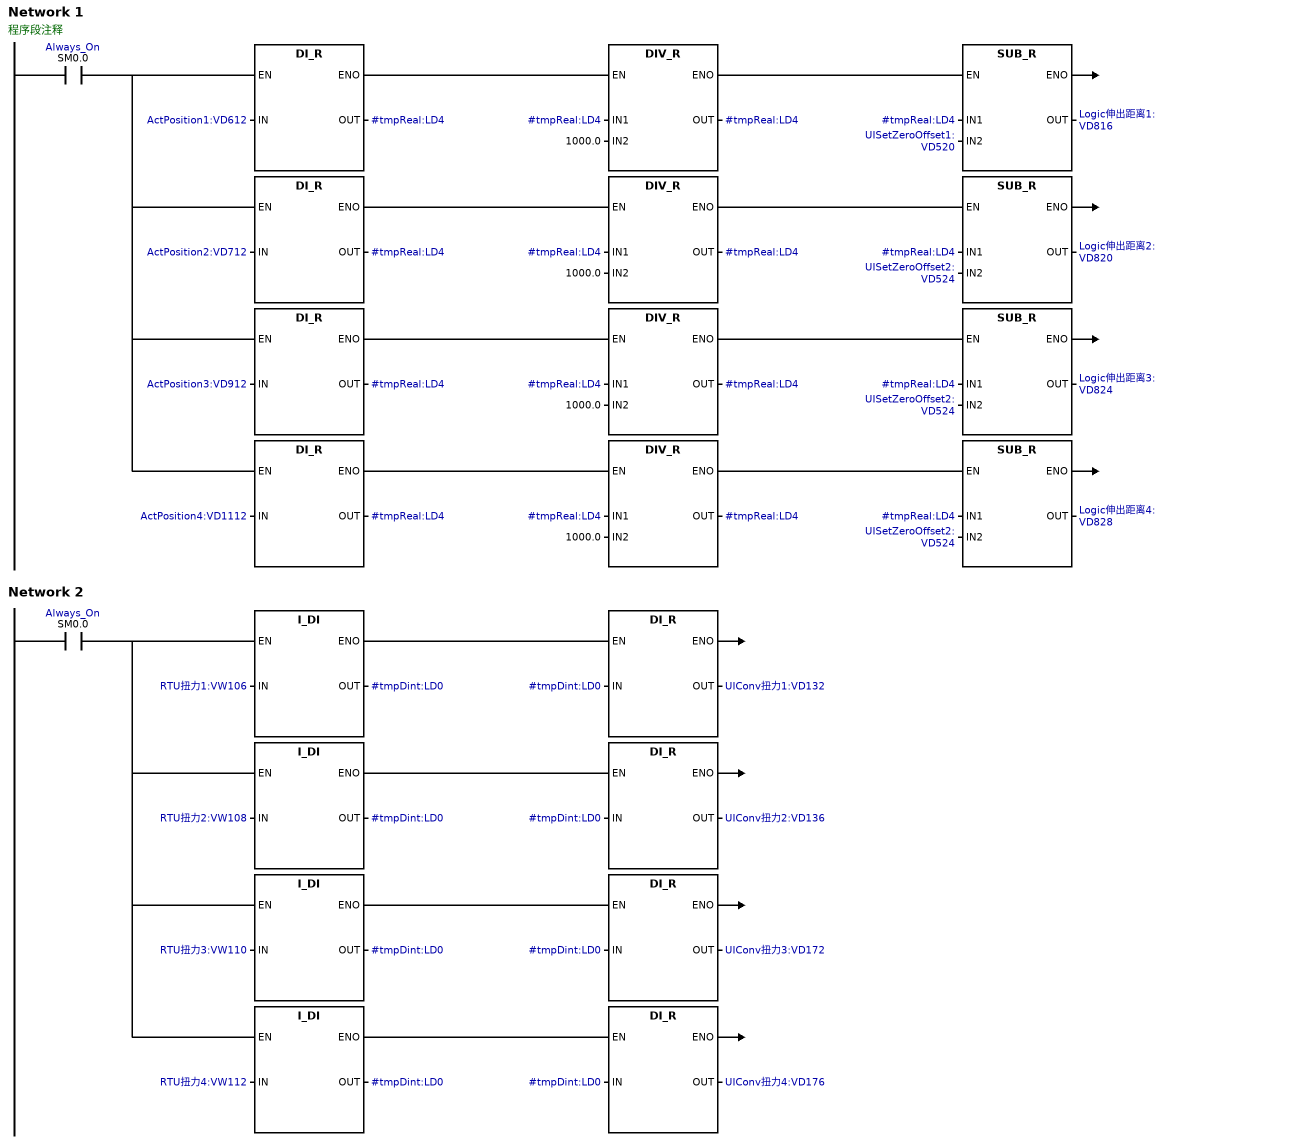
[picture p24: SBR6 networks 1-2]
Network 1
// 程序段注释
LD     Always_On:SM0.0
LPS
DTR    ActPosition1:VD612, #tmpReal:LD4
AENO
/R     1000.0, #tmpReal:LD4
AENO
MOVR   #tmpReal:LD4, Logic伸出距离1:VD816
-R     UISetZeroOffset1:VD520, Logic伸出距离1:VD816
LRD
DTR    ActPosition2:VD712, #tmpReal:LD4
AENO
/R     1000.0, #tmpReal:LD4
AENO
MOVR   #tmpReal:LD4, Logic伸出距离2:VD820
-R     UISetZeroOffset2:VD524, Logic伸出距离2:VD820
LRD
DTR    ActPosition3:VD912, #tmpReal:LD4
AENO
/R     1000.0, #tmpReal:LD4
AENO
MOVR   #tmpReal:LD4, Logic伸出距离3:VD824
-R     UISetZeroOffset2:VD524, Logic伸出距离3:VD824
LPP
DTR    ActPosition4:VD1112, #tmpReal:LD4
AENO
/R     1000.0, #tmpReal:LD4
AENO
MOVR   #tmpReal:LD4, Logic伸出距离4:VD828
-R     UISetZeroOffset2:VD524, Logic伸出距离4:VD828
Network 2
LD     Always_On:SM0.0
LPS
ITD    RTU扭力1:VW106, #tmpDint:LD0
AENO
DTR    #tmpDint:LD0, UIConv扭力1:VD132
LRD
ITD    RTU扭力2:VW108, #tmpDint:LD0
AENO
DTR    #tmpDint:LD0, UIConv扭力2:VD136
LRD
ITD    RTU扭力3:VW110, #tmpDint:LD0
AENO
DTR    #tmpDint:LD0, UIConv扭力3:VD172
LPP
ITD    RTU扭力4:VW112, #tmpDint:LD0
AENO
DTR    #tmpDint:LD0, UIConv扭力4:VD176
END_SUBROUTINE_BLOCK

// SBR7: protected block, not included

// SBR8: protected block, not included

SUBROUTINE_BLOCK XinJiePN:SBR9
TITLE=子程序注释
VAR
tmpSpeed:DWORD;	// LD0 
tmpPos1:DINT;	// LD4 
tmpWarning:WORD;	// LW8 
tmpErr:WORD;	// LW10 
tmpDone:BOOL;	// L12.0 
tmpNotJOD:BOOL;	// L12.1 
tmpPos2:DINT;	// LD13 
tmpReal:REAL;	// LD17 
tmpDint:DINT;	// LD21 
tmpPos3:DINT;	// LD25 
tmpPos4:DINT;	// LD29 
END_VAR
BEGIN
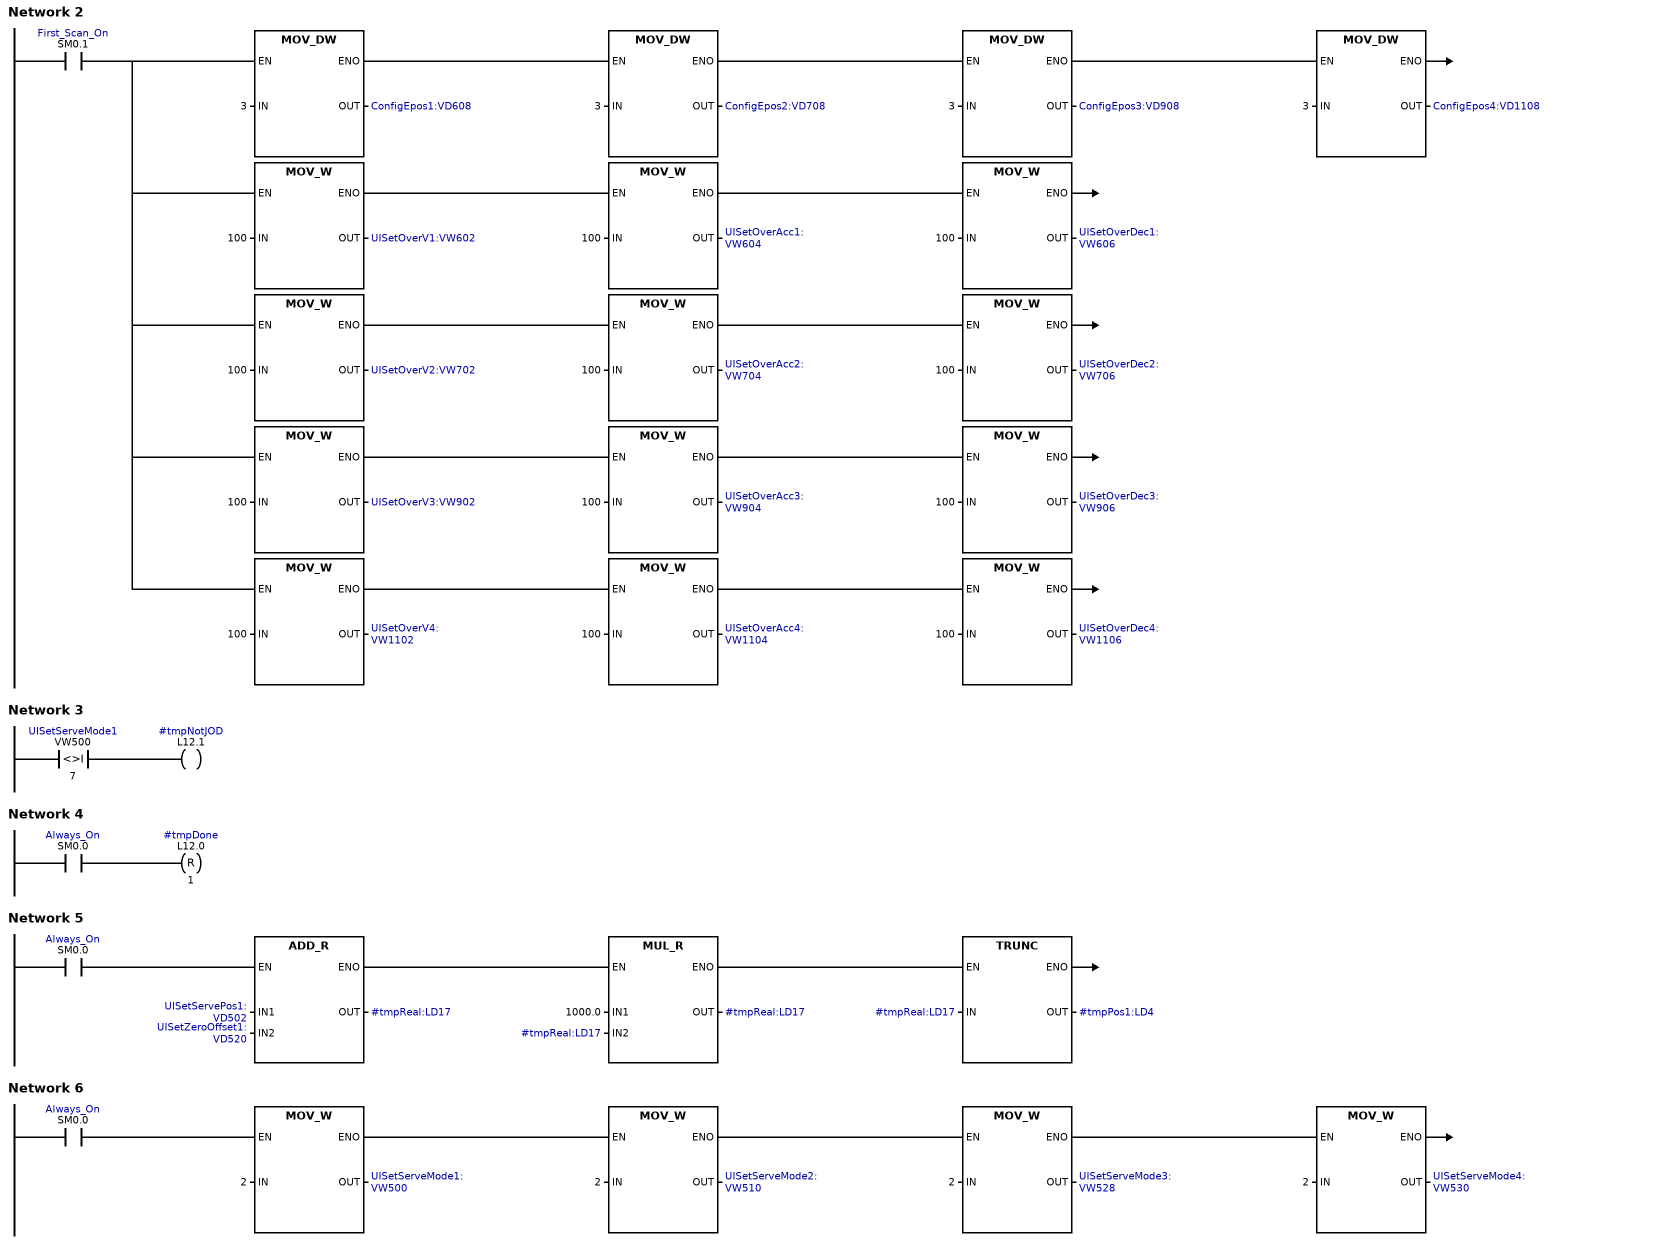
Network 2
LD     First_Scan_On:SM0.1
LPS
MOVD   3, ConfigEpos1:VD608
AENO
MOVD   3, ConfigEpos2:VD708
AENO
MOVD   3, ConfigEpos3:VD908
AENO
MOVD   3, ConfigEpos4:VD1108
LRD
MOVW   100, UISetOverV1:VW602
AENO
MOVW   100, UISetOverAcc1:VW604
AENO
MOVW   100, UISetOverDec1:VW606
LRD
MOVW   100, UISetOverV2:VW702
AENO
MOVW   100, UISetOverAcc2:VW704
AENO
MOVW   100, UISetOverDec2:VW706
LRD
MOVW   100, UISetOverV3:VW902
AENO
MOVW   100, UISetOverAcc3:VW904
AENO
MOVW   100, UISetOverDec3:VW906
LPP
MOVW   100, UISetOverV4:VW1102
AENO
MOVW   100, UISetOverAcc4:VW1104
AENO
MOVW   100, UISetOverDec4:VW1106
Network 3
LDW<>  UISetServeMode1:VW500, 7
=      #tmpNotJOD:L12.1
Network 4
LD     Always_On:SM0.0
R      #tmpDone:L12.0, 1
Network 5
LD     Always_On:SM0.0
MOVR   UISetServePos1:VD502, #tmpReal:LD17
AENO
+R     UISetZeroOffset1:VD520, #tmpReal:LD17
AENO
*R     1000.0, #tmpReal:LD17
AENO
TRUNC  #tmpReal:LD17, #tmpPos1:LD4
Network 6
LD     Always_On:SM0.0
MOVW   2, UISetServeMode1:VW500
AENO
MOVW   2, UISetServeMode2:VW510
AENO
MOVW   2, UISetServeMode3:VW528
AENO
MOVW   2, UISetServeMode4:VW530
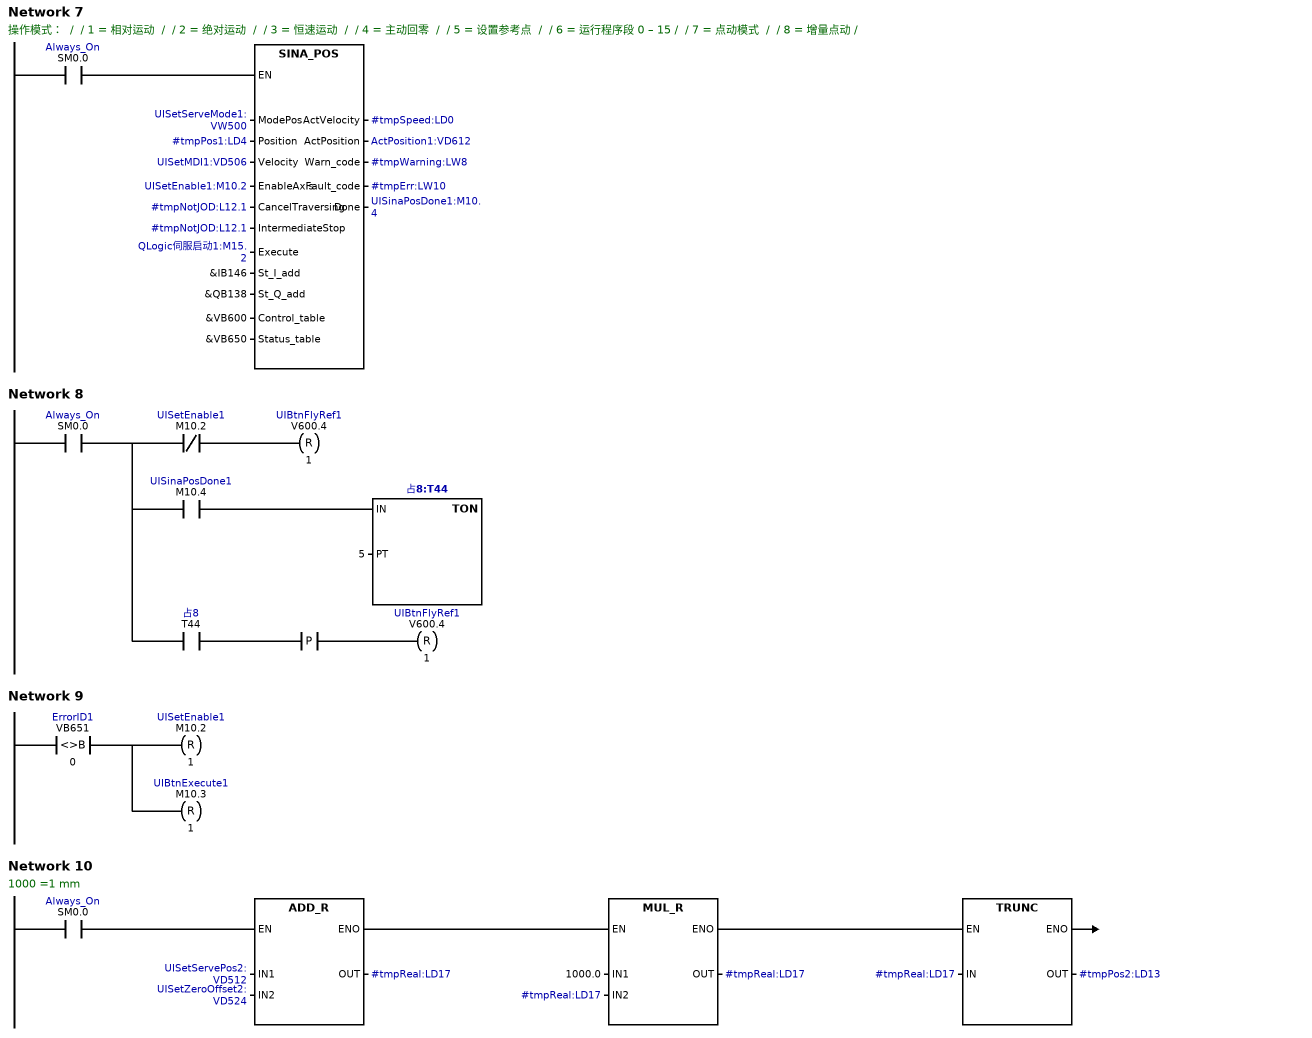
Network 7
// 操作模式： 
// 
// 1 = 相对运动 
// 
// 2 = 绝对运动 
// 
// 3 = 恒速运动 
// 
// 4 = 主动回零 
// 
// 5 = 设置参考点 
// 
// 6 = 运行程序段 0 – 15
// 
// 7 = 点动模式 
// 
// 8 = 增量点动
// 
LD     Always_On:SM0.0
CALL   SINA_POS:SBR8, UISetServeMode1:VW500, #tmpPos1:LD4, UISetMDI1:VD506, UISetEnable1:M10.2, #tmpNotJOD:L12.1, #tmpNotJOD:L12.1, QLogic伺服启动1:M15.2, &IB146, &QB138, &VB600, &VB650, #tmpSpeed:LD0, ActPosition1:VD612, #tmpWarning:LW8, #tmpErr:LW10, UISinaPosDone1:M10.4
Network 8
LD     Always_On:SM0.0
LPS
AN     UISetEnable1:M10.2
R      UIBtnFlyRef1:V600.4, 1
LRD
A      UISinaPosDone1:M10.4
TON    占8:T44, 5
LPP
A      占8:T44
EU
R      UIBtnFlyRef1:V600.4, 1
Network 9
LDB<>  ErrorID1:VB651, 0
R      UISetEnable1:M10.2, 1
R      UIBtnExecute1:M10.3, 1
Network 10
//  1000 =1 mm
LD     Always_On:SM0.0
MOVR   UISetServePos2:VD512, #tmpReal:LD17
AENO
+R     UISetZeroOffset2:VD524, #tmpReal:LD17
AENO
*R     1000.0, #tmpReal:LD17
AENO
TRUNC  #tmpReal:LD17, #tmpPos2:LD13
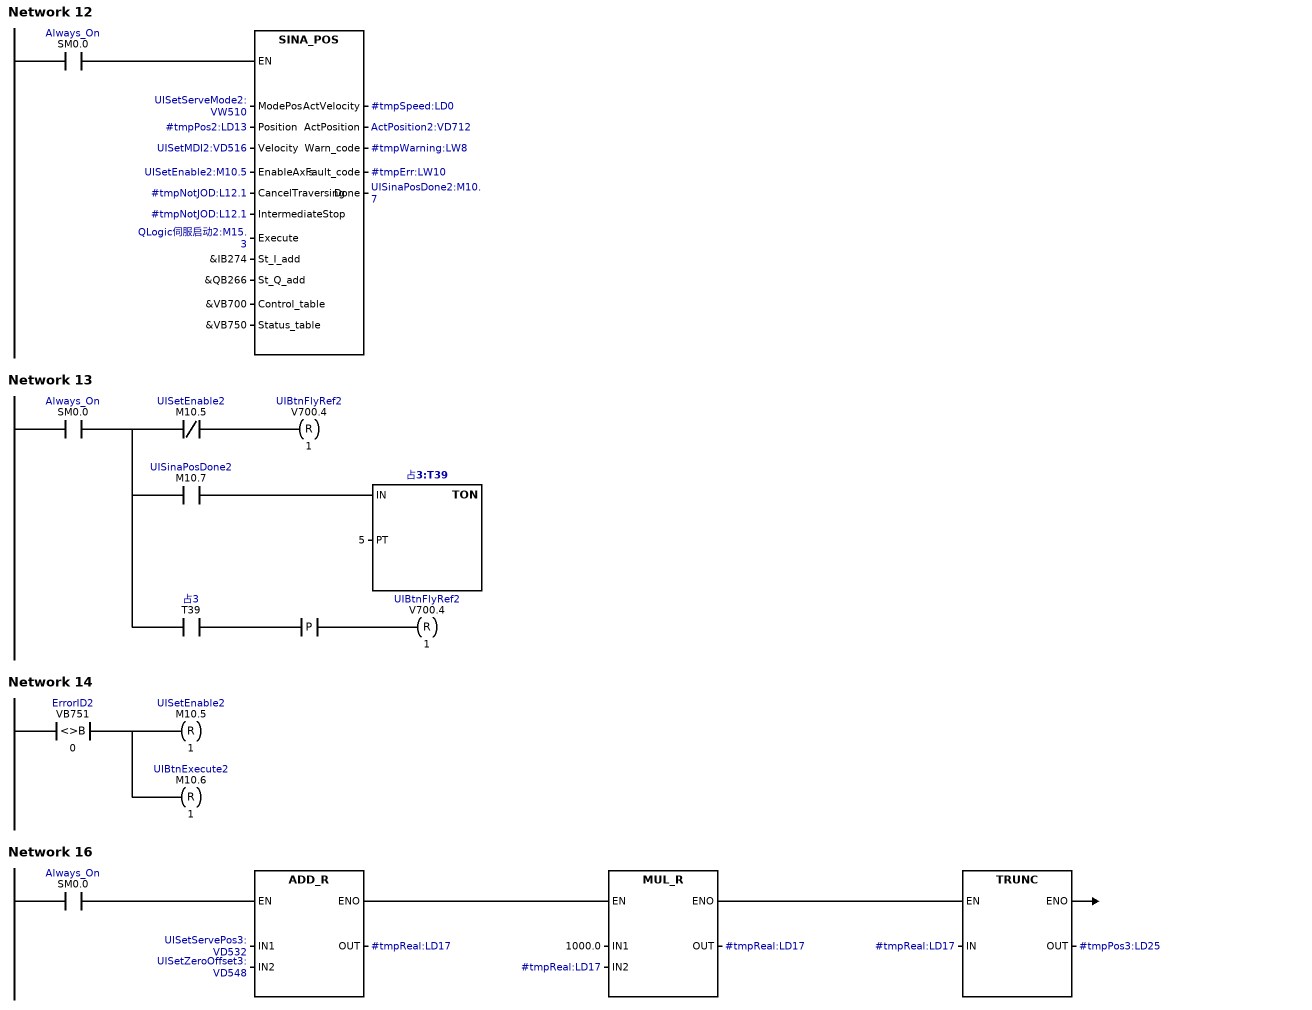
Network 12
LD     Always_On:SM0.0
CALL   SINA_POS:SBR8, UISetServeMode2:VW510, #tmpPos2:LD13, UISetMDI2:VD516, UISetEnable2:M10.5, #tmpNotJOD:L12.1, #tmpNotJOD:L12.1, QLogic伺服启动2:M15.3, &IB274, &QB266, &VB700, &VB750, #tmpSpeed:LD0, ActPosition2:VD712, #tmpWarning:LW8, #tmpErr:LW10, UISinaPosDone2:M10.7
Network 13
LD     Always_On:SM0.0
LPS
AN     UISetEnable2:M10.5
R      UIBtnFlyRef2:V700.4, 1
LRD
A      UISinaPosDone2:M10.7
TON    占3:T39, 5
LPP
A      占3:T39
EU
R      UIBtnFlyRef2:V700.4, 1
Network 14
LDB<>  ErrorID2:VB751, 0
R      UISetEnable2:M10.5, 1
R      UIBtnExecute2:M10.6, 1
Network 16
LD     Always_On:SM0.0
MOVR   UISetServePos3:VD532, #tmpReal:LD17
AENO
+R     UISetZeroOffset3:VD548, #tmpReal:LD17
AENO
*R     1000.0, #tmpReal:LD17
AENO
TRUNC  #tmpReal:LD17, #tmpPos3:LD25
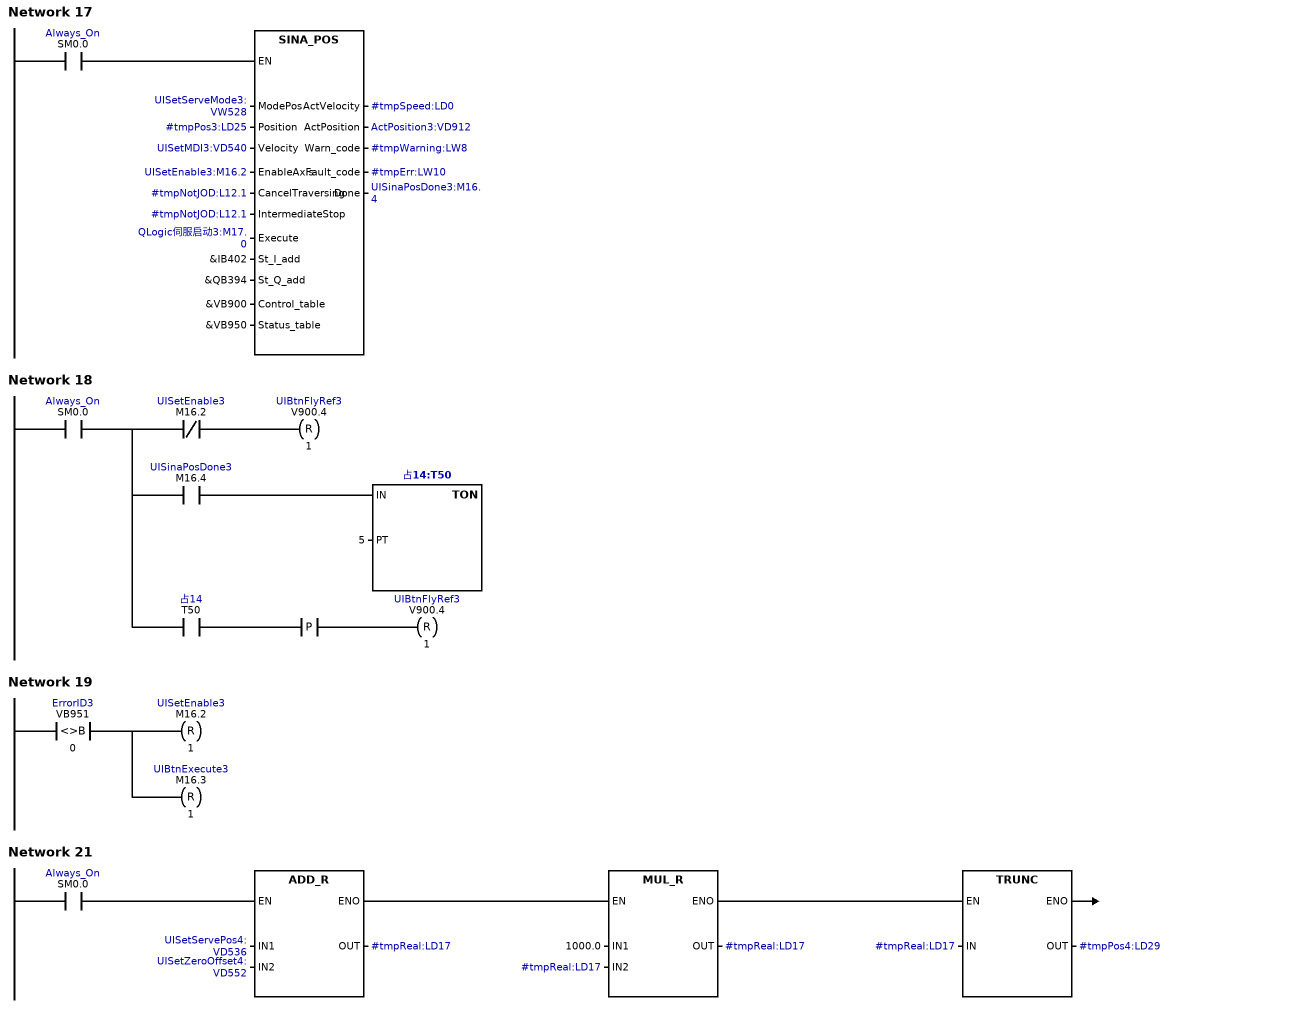
Network 17
LD     Always_On:SM0.0
CALL   SINA_POS:SBR8, UISetServeMode3:VW528, #tmpPos3:LD25, UISetMDI3:VD540, UISetEnable3:M16.2, #tmpNotJOD:L12.1, #tmpNotJOD:L12.1, QLogic伺服启动3:M17.0, &IB402, &QB394, &VB900, &VB950, #tmpSpeed:LD0, ActPosition3:VD912, #tmpWarning:LW8, #tmpErr:LW10, UISinaPosDone3:M16.4
Network 18
LD     Always_On:SM0.0
LPS
AN     UISetEnable3:M16.2
R      UIBtnFlyRef3:V900.4, 1
LRD
A      UISinaPosDone3:M16.4
TON    占14:T50, 5
LPP
A      占14:T50
EU
R      UIBtnFlyRef3:V900.4, 1
Network 19
LDB<>  ErrorID3:VB951, 0
R      UISetEnable3:M16.2, 1
R      UIBtnExecute3:M16.3, 1
Network 21
LD     Always_On:SM0.0
MOVR   UISetServePos4:VD536, #tmpReal:LD17
AENO
+R     UISetZeroOffset4:VD552, #tmpReal:LD17
AENO
*R     1000.0, #tmpReal:LD17
AENO
TRUNC  #tmpReal:LD17, #tmpPos4:LD29
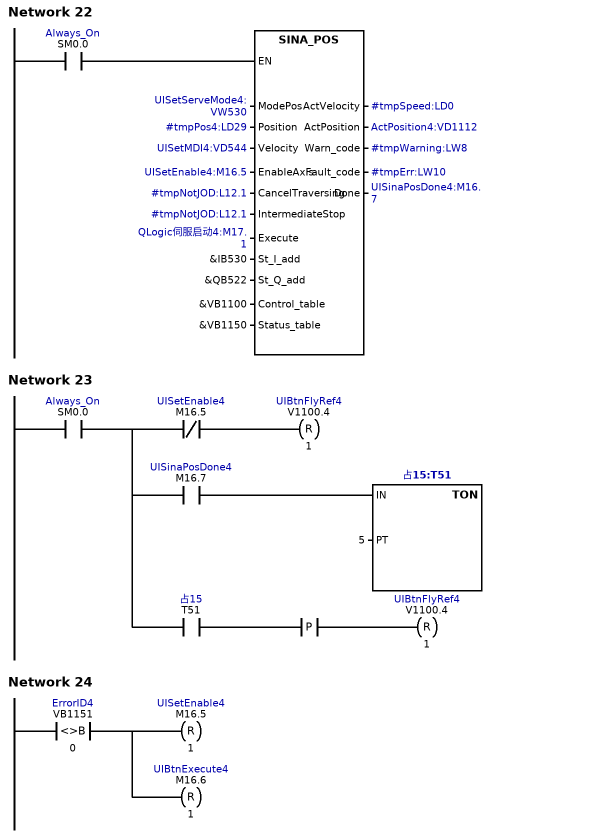
Network 22
LD     Always_On:SM0.0
CALL   SINA_POS:SBR8, UISetServeMode4:VW530, #tmpPos4:LD29, UISetMDI4:VD544, UISetEnable4:M16.5, #tmpNotJOD:L12.1, #tmpNotJOD:L12.1, QLogic伺服启动4:M17.1, &IB530, &QB522, &VB1100, &VB1150, #tmpSpeed:LD0, ActPosition4:VD1112, #tmpWarning:LW8, #tmpErr:LW10, UISinaPosDone4:M16.7
Network 23
LD     Always_On:SM0.0
LPS
AN     UISetEnable4:M16.5
R      UIBtnFlyRef4:V1100.4, 1
LRD
A      UISinaPosDone4:M16.7
TON    占15:T51, 5
LPP
A      占15:T51
EU
R      UIBtnFlyRef4:V1100.4, 1
Network 24
LDB<>  ErrorID4:VB1151, 0
R      UISetEnable4:M16.5, 1
R      UIBtnExecute4:M16.6, 1
END_SUBROUTINE_BLOCK

// SBR10: protected block, not included

// SBR11: protected block, not included

// SBR12: protected block, not included
